FUNCTION Convert_UDINT_TO_LINT : BOOL
VAR_INPUT
	in : UDINT;
	out : REFERENCE TO LINT;
END_VAR
VAR
	converted : LINT;
END_VAR

converted := UDINT_TO_LINT(in);

IF (LINT_TO_UDINT(converted) <> in) THEN
	RETURN;
END_IF

out := converted;
Convert_UDINT_TO_LINT := TRUE;

END_FUNCTION

(* stored: Version 1.1.0.1, ProductVersion 3.1.4024.12
   POU Convert_UDINT_TO_LINT: Id {8d689b22-aeb7-4fac-90ad-a9918e1ff9b7}, SpecialFunc None *)
